FUNCTION_BLOCK Monitor
  (* Standard: 61499-2 *)
  (* Version 0.2, 2003-12-04, JHC, Rockwell Automation, Renamed for better indexing. *)
  (* Version 0.1, 2002-11-05, JHC, Rockwell Automation, Corrected missing ST element in Algorithm REQ. *)
  (* Version 0.0, 2000-05-30, JHC, Rockwell Automation *)
  (* Compiler header: package fb.rt.benchmarks.watermonitor; *)
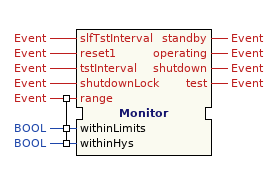
  EVENT_INPUT
    slfTstInterval;
    reset1;
    tstInterval;
    shutdownLock;
    range WITH withinLimits, withinHys;
  END_EVENT
  EVENT_OUTPUT
    standby;
    operating;
    shutdown;
    test;
  END_EVENT
  VAR_INPUT
    withinLimits : BOOL := true;
    withinHys : BOOL := true;
  END_VAR
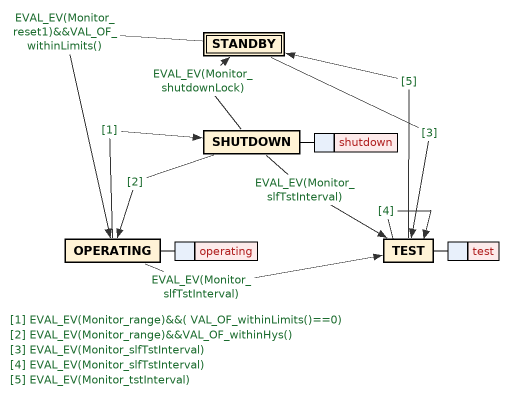
  EC_STATES
    STANDBY; (* Initial State *)
    SHUTDOWN : -> shutdown;
    OPERATING : -> operating;
    TEST : -> test;
  END_STATES
  EC_TRANSITIONS
    STANDBY TO TEST := EVAL_EV(Monitor_slfTstInterval);
    STANDBY TO OPERATING := EVAL_EV(Monitor_reset1)&&VAL_OF_withinLimits();
    TEST TO TEST := EVAL_EV(Monitor_slfTstInterval);
    TEST TO STANDBY := EVAL_EV(Monitor_tstInterval);
    OPERATING TO TEST := EVAL_EV(Monitor_slfTstInterval);
    OPERATING TO SHUTDOWN := EVAL_EV(Monitor_range)&&( VAL_OF_withinLimits()==0);
    SHUTDOWN TO TEST := EVAL_EV(Monitor_slfTstInterval);
    SHUTDOWN TO OPERATING := EVAL_EV(Monitor_range)&&VAL_OF_withinHys();
    SHUTDOWN TO STANDBY := EVAL_EV(Monitor_shutdownLock);
  END_TRANSITIONS
END_FUNCTION_BLOCK
